INTERFACE I_HomeDS402 EXTENDS I_Home

{warning 'Add property implementation'}
PROPERTY CommandMoveHome : BOOL
SET
END_SET
END_PROPERTY

PROPERTY ControlWord : UINT
GET
END_GET
END_PROPERTY

PROPERTY Mode : E_EpicsHomeCmd
GET
END_GET
SET
END_SET
END_PROPERTY

PROPERTY ModeOfOperation : SINT
GET
END_GET
END_PROPERTY

{warning 'Add property implementation'}
PROPERTY Offset : LREAL
SET
END_SET
END_PROPERTY

{warning 'Add property implementation'}
PROPERTY Position : LREAL
SET
END_SET
END_PROPERTY

METHOD Status
VAR_INPUT
	ModeOfOperationDisplay : SINT;
	Bit13OpModeSpecific	: BOOL;
	Bit12OpModeSpecific	: BOOL;
	TargetReached	: BOOL;
END_VAR
END_METHOD

END_INTERFACE

(* stored: Version 1.1.0.1
   Itf I_HomeDS402: Id {7f1d3075-62c7-47b5-b35e-42b4971857a7}
   Property CommandMoveHome: Id {0e532e9d-38ed-40b8-81b0-3a8c690b9bb4}
   Set Set: Id {137fcfe1-22e4-4e29-bc47-b7daad71e451}
   Property ControlWord: Id {758d5033-e1d3-4a22-b240-f5626aa91569}
   Get Get: Id {ebeda8d8-3f26-4ec1-b4b8-3d18303b5531}
   Property Mode: Id {a3c276b4-a4a3-4cbf-a4ae-ec2cedfa8435}
   Get Get: Id {ccb0abb4-4d0f-4d51-b517-165ca4ae30c2}
   Set Set: Id {725ce957-0a17-40d3-b82b-8f5bd85c42ec}
   Property ModeOfOperation: Id {17fbe6d4-257a-4d8e-a349-fd82e025b222}
   Get Get: Id {90e68fe1-fb52-4c6b-b8c9-baf2da28495c}
   Property Offset: Id {dfdec895-8f5a-4a35-9dee-19e76ad604c0}
   Set Set: Id {d4a1a429-33e0-4d3f-a309-9e0961aa87f0}
   Property Position: Id {166022b2-e85d-404e-87c1-c2161b43adfb}
   Set Set: Id {7de22104-8291-4fdd-9b16-e078d4d41d8a}
   Method Status: Id {a53b6c8c-96e3-4eb0-9dd0-0ee54d847836} *)
